Staubli VAL3: loadCycle.pgx

public program loadCycle(string& x_sName[], num& x_nResult[])
begin
  //
  // load the select program for the Cycle
  //
end
